SUBAPPLICATION Uebung_073_AUI (* VDS auf UT ausgeben (Adapter Version) *)
  (* Standard: 61499-2; Description: Copyright (c) 2023 Meisterschulen am Ostbahnhof This program and the accompanying materials are made available under the terms of the Eclipse Public License 2.0 which is available at https://www.eclipse.org/legal/epl-2.0/ SPDX-License-Identifier: EPL-2.0 *)
  (* Version 1.0, 2026-04-19, Franz Höpfinger, Meisterschulen am Ostbahnhof, initial API and implementation (Adapter Version of Uebung_073) *)
  PACKAGE Uebungen;
  IMPORT Uebungen::const::UT::TECU::DefaultPool_TECU::NumberVariable_Wheel_based_machine_speed;
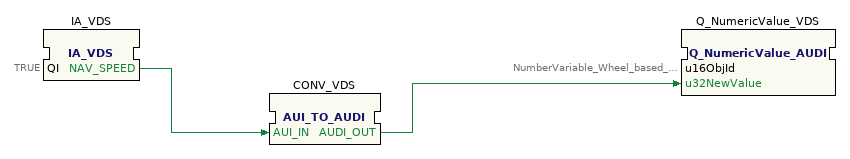
  FBS
    IA_VDS : isobus::tecu::IA_VDS(QI := TRUE);
    Q_NumericValue_VDS : isobus::UT::Q::Q_NumericValue_AUDI(u16ObjId := NumberVariable_Wheel_based_machine_speed);
    CONV_VDS : adapter::conversion::unidirectional::AUI_TO_AUDI;
  END_FBS
  ADAPTER_CONNECTIONS
    IA_VDS.NAV_SPEED TO CONV_VDS.AUI_IN;
    CONV_VDS.AUDI_OUT TO Q_NumericValue_VDS.u32NewValue;
  END_CONNECTIONS
END_SUBAPPLICATION
